// TwinCAT 3 PLC project PlcIotHttpSamplesPostman
// ProgramVersion: 3.1.4026.25
// libraries:
//   Tc2_Standard, * (Beckhoff Automation GmbH)
//   Tc2_System, * (Beckhoff Automation GmbH)
//   Tc2_Utilities, * (Beckhoff Automation GmbH)
//   Tc3_IotBase, * (Beckhoff Automation GmbH)
//   Tc3_JsonXml, * (Beckhoff Automation GmbH)
//   Tc3_Module, * (Beckhoff Automation GmbH)
// project tree:
//   / PlcTask.TcTTO (not stored)
//   POUs/ MAIN.TcPOU
//   POUs/Postman/ FB_TestHTTP_Get.TcPOU, FB_TestHTTP_HeaderAuth.TcPOU, FB_TestHTTP_Post.TcPOU, FB_TestHTTP_Put.TcPOU
// real-time tasks:
//   TASK PlcTask: cycle T#10ms, priority 21, ADS port 350

// ---- POUs/MAIN.TcPOU
PROGRAM MAIN
VAR
	// trigger command execution for Postman-Echo samples
	bGet, bPost, bPut, bHeaderAuth 	: BOOL;

	fbHttpClientPostman				: FB_IotHttpClient :=(sHostName := 'postman-echo.com',
								  	bKeepAlive := TRUE, tConnectionTimeout := T#10S);
								
	fbHttpGet						: FB_TestHTTP_Get;
	fbHttpPost						: FB_TestHTTP_Post;
	fbHttpPut						: FB_TestHTTP_Put;
	fbHttpHeaderAuth				: FB_TestHTTP_HeaderAuth;
END_VAR

// init client parameters at startup
IF NOT fbHttpClientPostman.bConfigured THEN 
	fbHttpClientPostman.nHostPort := 443;
	fbHttpClientPostman.stTLS.bNoServerCertCheck := TRUE;
END_IF

IF fbHttpClientPostman.bConfigured THEN 
	fbHttpGet(bSend := bGet, fbClient := fbHttpClientPostman);
	fbHttpPost(bSend := bPost, fbClient := fbHttpClientPostman);
	fbHttpPut(bSend := bPut, fbClient := fbHttpClientPostman);
	fbHttpHeaderAuth(bSend := bHeaderAuth, fbClient := fbHttpClientPostman);
END_IF 

fbHttpClientPostman.Execute();

END_PROGRAM

// ---- POUs/Postman/FB_TestHTTP_Get.TcPOU
FUNCTION_BLOCK FB_TestHTTP_Get
VAR_INPUT
	bSend				: BOOL;
END_VAR
VAR_IN_OUT
	fbClient			: FB_IotHttpClient;
END_VAR
VAR_OUTPUT
	bBusy				: BOOL;
	bError				: BOOL;
END_VAR
VAR
	fbRequest			: FB_IotHttpRequest;
	fbJson				: FB_JsonDomParser;
	nState				: UDINT;
	RisingEdge			: R_TRIG;
	
	bGetContentResult	: BOOL;
	sContent			: STRING(511);
	
	bGetJsonResult		: BOOL;
	jsonDoc				: SJsonValue;
	jsonVal				: SJsonValue;
	sResultValue		: STRING;
	
	nReqCount			: UDINT;	
	nResCount			: UDINT;
	nValidResCount		: UDINT;
	nErrCount			: UDINT;
END_VAR

RisingEdge(CLK := bSend );
CASE nState OF
0:	
	IF RisingEdge.Q THEN 
		IF fbRequest.SendRequest(sUri := '/get?foo1=bar1&foo2=bar2', fbClient := fbClient, eRequestType := ETcIotHttpRequestType.HTTP_GET, 0, 0, 0) THEN				
			nState := 1;
			nReqCount := nReqCount +1;
			bBusy := TRUE;
			bError := FALSE;
		END_IF					
	END_IF
1:
	IF NOT fbRequest.bBusy THEN
		bError := TRUE;
		IF NOT fbRequest.bError THEN
			// As an alternative to GetJsonDomContent, GetContent could be used				 
			// bGetContentResult := fbRequest.GetContent(pContent := ADR(sContent), nContentSize := SIZEOF(sContent), bSetNullTermination := TRUE);
			IF fbRequest.nStatusCode >= 200 AND fbRequest.nStatusCode < 300 THEN
				bGetJsonResult := FALSE;
				// Direct conversion into JSON object as the received message is in JSON format 
				jsonDoc := fbRequest.GetJsonDomContent(fbJson);
				IF jsonDoc <> 0 THEN
					bGetJsonResult := TRUE;
					IF fbJson.HasMember(jsonDoc, 'args')  THEN
						jsonVal := fbJson.FindMember(jsonDoc, 'args');
						IF fbJson.HasMember(jsonVal, 'foo2')  THEN
							jsonVal := fbJson.FindMember(jsonVal, 'foo2');
							bError := FALSE;						
							IF fbJson.IsString(jsonVal) THEN						
								sResultValue := fbJson.GetString(jsonVal);
								IF sResultValue = 'bar2' THEN
									// Received STRING value must be bar2
									nValidResCount := nValidResCount +1;
								END_IF							
							END_IF
						END_IF		
					END_IF
				END_IF							
				nResCount := nResCount +1;			
			END_IF
		END_IF
		nState := 0;
		bBusy := FALSE;
		IF bError THEN
			nErrCount := nErrCount +1;
		END_IF
	END_IF  	
END_CASE

END_FUNCTION_BLOCK

// ---- POUs/Postman/FB_TestHTTP_Post.TcPOU
FUNCTION_BLOCK FB_TestHTTP_Post
VAR_INPUT
	bSend				: BOOL;
END_VAR
VAR_IN_OUT
	fbClient			: FB_IotHttpClient;
END_VAR
VAR_OUTPUT
	bBusy				: BOOL;
	bError				: BOOL;
END_VAR
VAR	
	fbRequest			: FB_IotHttpRequest;
	fbJson				: FB_JsonDomParser;
	nState				: UDINT;
	RisingEdge			: R_TRIG;
	
	bGetContentResult	: BOOL;
	sContent			: STRING(511);
	
	bGetJsonResult		: BOOL;
	jsonDoc				: SJsonValue;
	jsonVal				: SJsonValue;
	sResultValue		: STRING;
	
	nReqCount			: UDINT;
	nResCount			: UDINT;
	nValidResCount		: UDINT;
	nErrCount			: UDINT;	
END_VAR

RisingEdge(CLK := bSend);
CASE nState OF
0:		
	IF RisingEdge.Q THEN 
		sContent := 'This is some sample HTTP POST content';
		IF fbRequest.SendRequest(sUri:= '/post?hello=world', fbClient := fbClient, eRequestType := ETcIotHttpRequestType.HTTP_POST, pContent := ADR(sContent), nContentSize := LEN2(ADR(sContent)), 0) THEN				
			nState := 1;
			nReqCount := nReqCount +1;
			bBusy := TRUE;
			bError := FALSE;
		END_IF					
	END_IF
1:
	IF NOT fbRequest.bBusy THEN
		bError := TRUE;
		IF NOT fbRequest.bError THEN				 				
			// As an alternative to GetJsonDomContent, GetContent could be used				 
			// bGetContentResult := fbRequest.GetContent(pContent := ADR(sContent), nContentSize := SIZEOF(sContent), bSetNullTermination := TRUE);
			IF fbRequest.nStatusCode >= 200 AND fbRequest.nStatusCode < 300 THEN
				bGetJsonResult := FALSE;
				// Direct conversion into JSON object as the received message is in JSON format 
				jsonDoc := fbRequest.GetJsonDomContent(fbJson);				
				IF jsonDoc <> 0 THEN
					bGetJsonResult := TRUE;
					IF fbJson.HasMember(jsonDoc, 'data')  THEN
						jsonVal := fbJson.FindMember(jsonDoc, 'data');
						sResultValue := fbJson.GetString(jsonVal);
						IF sResultValue = sContent THEN
							// Received value has to be equal with sent value
							nValidResCount := nValidResCount +1;
							bError := FALSE;
						END_IF
					END_IF		
				END_IF
				nResCount := nResCount +1;					
			END_IF				
		END_IF
		nState := 0;
		bBusy := FALSE;
		IF bError THEN
			nErrCount := nErrCount +1;
		END_IF		
	END_IF  	
END_CASE

END_FUNCTION_BLOCK

// ---- POUs/Postman/FB_TestHTTP_Put.TcPOU
FUNCTION_BLOCK FB_TestHTTP_Put
VAR_INPUT
	bSend				: BOOL;
END_VAR
VAR_IN_OUT
	fbClient			: FB_IotHttpClient;
END_VAR
VAR_OUTPUT
	bBusy				: BOOL;
	bError				: BOOL;
END_VAR
VAR	
	fbRequest			: FB_IotHttpRequest;
	fbJson				: FB_JsonDomParser;
	nState				: UDINT;
	RisingEdge			: R_TRIG;
	
	bGetContentResult	: BOOL;
	sContent			: STRING(511);
	
	bGetJsonResult		: BOOL;
	jsonDoc				: SJsonValue;
	jsonVal				: SJsonValue;
	sResultValue		: STRING;
		
	nReqCount			: UDINT;
	nResCount			: UDINT;
	nValidResCount		: UDINT;
	nErrCount			: UDINT;	
END_VAR

RisingEdge(CLK := bSend);
CASE nState OF
0:		
	IF RisingEdge.Q THEN 
		sContent := 'This is some sample HTTP PUT content';
		IF fbRequest.SendRequest(sUri := '/put', fbClient := fbClient, eRequestType := ETcIotHttpRequestType.HTTP_PUT, pContent := ADR(sContent), nContentSize := LEN2(ADR(sContent)), 0) THEN				
			nState := 1;
			nReqCount := nReqCount +1;
			bBusy := TRUE;
			bError := FALSE;
		END_IF
	END_IF
1:
	IF NOT fbRequest.bBusy THEN
		bError := TRUE;
		IF NOT fbRequest.bError THEN				 
			// As an alternative to GetJsonDomContent, GetContent could be used				 
			// bGetContentResult := fbRequest.GetContent(pContent := ADR(sContent), nContentSize := SIZEOF(sContent), bSetNullTermination := TRUE);	
			IF fbRequest.nStatusCode >= 200 AND fbRequest.nStatusCode < 300 THEN
				bGetJsonResult := FALSE;
				// Direct conversion into JSON object as the received message is in JSON format 
				jsonDoc := fbRequest.GetJsonDomContent(fbJson);				
				IF jsonDoc <> 0 THEN
					bGetJsonResult := TRUE;
					IF fbJson.HasMember(jsonDoc, 'data')  THEN
						jsonVal := fbJson.FindMember(jsonDoc, 'data');
						sResultValue := fbJson.GetString(jsonVal);
						IF sResultValue = sContent THEN
							// Received value has to be equal with sent value
							nValidResCount := nValidResCount +1;
							bError := FALSE;
						END_IF
					END_IF	
				END_IF					
				nResCount := nResCount +1;					
			END_IF				
		END_IF
		nState := 0;
		bBusy := FALSE;
		IF bError THEN
			nErrCount := nErrCount +1;
		END_IF		
	END_IF  	
END_CASE

END_FUNCTION_BLOCK

// ---- POUs/Postman/FB_TestHTTP_HeaderAuth.TcPOU
FUNCTION_BLOCK FB_TestHTTP_HeaderAuth
VAR_INPUT
	bSend		: BOOL;
END_VAR
VAR_IN_OUT
	fbClient			: FB_IotHttpClient;
END_VAR
VAR_OUTPUT
	bBusy				: BOOL;
	bError				: BOOL;
END_VAR
VAR
	fbRequest			: FB_IotHttpRequest;
	fbHeader			: FB_IotHttpHeaderFieldMap;
	fbJson				: FB_JsonDomParser;
	nState				: UDINT;
	RisingEdge			: R_TRIG;

	bGetContentResult	: BOOL;
	sContent			: STRING(511);
	
	bGetJsonResult		: BOOL;
	jsonDoc				: SJsonValue;
	jsonVal				: SJsonValue;
	bResultValue		: BOOL;
	
	nReqCount			: UDINT;	
	nResCount			: UDINT;
	nValidResCount		: UDINT;
	nErrCount			: UDINT;
	bOnce				: BOOL:= TRUE;
END_VAR

IF bOnce THEN
	fbHeader.AddField('Authorization', 'Basic cG9zdG1hbjpwYXNzd29yZA==', FALSE);	
	bOnce := FALSE;
END_IF

RisingEdge(CLK := bSend);
CASE nState OF
0:	
	IF RisingEdge.Q THEN 
		IF fbRequest.SendRequest(sUri := '/basic-auth', fbClient := fbClient, eRequestType := ETcIotHttpRequestType.HTTP_GET, 0, 0, fbHeader) THEN				
			nState := 1;
			nReqCount := nReqCount+1;
			bBusy := TRUE;
			bError := FALSE;
		END_IF					
	END_IF
1:
	IF NOT fbRequest.bBusy THEN
		bError := TRUE;
		IF NOT fbRequest.bError THEN				 
			// As an alternative to GetJsonDomContent, GetContent could be used				 
			// bGetContentResult := fbRequest.GetContent(pContent := ADR(sContent), nContentSize := SIZEOF(sContent), bSetNullTermination := TRUE);
			IF fbRequest.nStatusCode >= 200 AND fbRequest.nStatusCode < 300 THEN
				bGetJsonResult := FALSE;				
				// Direct conversion into JSON object as the received message is in JSON format 
				jsonDoc := fbRequest.GetJsonDomContent(fbJson);
				IF jsonDoc <> 0 THEN
					bGetJsonResult := TRUE;
					IF fbJson.HasMember(jsonDoc, 'authenticated') THEN
						jsonVal := fbJson.FindMember(jsonDoc, 'authenticated');						
						IF fbJson.IsBool(jsonVal) THEN
							// Value is TRUE when authentication worked correctly
							bResultValue := fbJson.GetBool(jsonVal);
							nValidResCount := nValidResCount +1;
							bError := FALSE;						
						END_IF	
					END_IF
				END_IF							
				nResCount := nResCount +1;			
			END_IF
		END_IF
		nState := 0;
		bBusy := FALSE;
		IF bError THEN
			nErrCount := nErrCount +1;
		END_IF
	END_IF  	
END_CASE

END_FUNCTION_BLOCK
